FUNCTION_BLOCK EC_SENSORS_ACTUATORS (* Composite Function Block Type *)
  (* Standard: 61499-2 *)
  (* Version 1.0, 2019-03-30, adeel *)
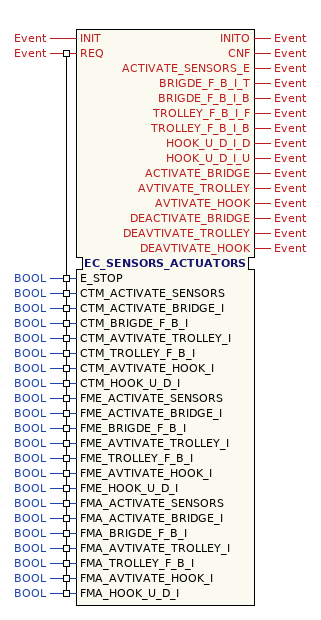
  EVENT_INPUT
    INIT; (* Initialization Request *)
    REQ WITH CTM_ACTIVATE_SENSORS, CTM_ACTIVATE_BRIDGE_I, CTM_BRIGDE_F_B_I, CTM_AVTIVATE_TROLLEY_I, CTM_TROLLEY_F_B_I, CTM_AVTIVATE_HOOK_I, CTM_HOOK_U_D_I, FME_ACTIVATE_SENSORS, FME_ACTIVATE_BRIDGE_I, FME_BRIGDE_F_B_I, FME_AVTIVATE_TROLLEY_I, FME_TROLLEY_F_B_I, FME_AVTIVATE_HOOK_I, FME_HOOK_U_D_I, FMA_ACTIVATE_SENSORS, FMA_ACTIVATE_BRIDGE_I, FMA_BRIGDE_F_B_I, FMA_AVTIVATE_TROLLEY_I, FMA_TROLLEY_F_B_I, FMA_AVTIVATE_HOOK_I, FMA_HOOK_U_D_I, E_STOP; (* Normal Execution Request *)
  END_EVENT
  EVENT_OUTPUT
    INITO; (* Initialization Confirm *)
    CNF;
    ACTIVATE_SENSORS_E;
    BRIGDE_F_B_I_T;
    BRIGDE_F_B_I_B;
    TROLLEY_F_B_I_F;
    TROLLEY_F_B_I_B;
    HOOK_U_D_I_D;
    HOOK_U_D_I_U;
    ACTIVATE_BRIDGE;
    AVTIVATE_TROLLEY;
    AVTIVATE_HOOK;
    DEACTIVATE_BRIDGE;
    DEAVTIVATE_TROLLEY;
    DEAVTIVATE_HOOK;
  END_EVENT
  VAR_INPUT
    E_STOP : BOOL;
    CTM_ACTIVATE_SENSORS : BOOL;
    CTM_ACTIVATE_BRIDGE_I : BOOL;
    CTM_BRIGDE_F_B_I : BOOL;
    CTM_AVTIVATE_TROLLEY_I : BOOL;
    CTM_TROLLEY_F_B_I : BOOL;
    CTM_AVTIVATE_HOOK_I : BOOL;
    CTM_HOOK_U_D_I : BOOL;
    FME_ACTIVATE_SENSORS : BOOL;
    FME_ACTIVATE_BRIDGE_I : BOOL;
    FME_BRIGDE_F_B_I : BOOL;
    FME_AVTIVATE_TROLLEY_I : BOOL;
    FME_TROLLEY_F_B_I : BOOL;
    FME_AVTIVATE_HOOK_I : BOOL;
    FME_HOOK_U_D_I : BOOL;
    FMA_ACTIVATE_SENSORS : BOOL;
    FMA_ACTIVATE_BRIDGE_I : BOOL;
    FMA_BRIGDE_F_B_I : BOOL;
    FMA_AVTIVATE_TROLLEY_I : BOOL;
    FMA_TROLLEY_F_B_I : BOOL;
    FMA_AVTIVATE_HOOK_I : BOOL;
    FMA_HOOK_U_D_I : BOOL;
  END_VAR
  FBS
    CTM_11 : E_R_TRIG;
    CTM_12 : E_F_TRIG;
    CTM_21 : E_R_TRIG;
    CTM_22 : E_F_TRIG;
    CTM_31 : E_R_TRIG;
    CTM_32 : E_F_TRIG;
    CTM_41 : E_R_TRIG;
    CTM_42 : E_F_TRIG;
    FME41 : E_R_TRIG;
    FME_11 : E_R_TRIG;
    FME_32 : E_F_TRIG;
    FME_42 : E_F_TRIG;
    FME_31 : E_R_TRIG;
    FME_12 : E_F_TRIG;
    FME_21 : E_R_TRIG;
    FME_22 : E_F_TRIG;
    FMA_41 : E_R_TRIG;
    FMA_11 : E_R_TRIG;
    FMA_32 : E_F_TRIG;
    FMA_42 : E_F_TRIG;
    FMA_31 : E_R_TRIG;
    FMA_12 : E_F_TRIG;
    FMA_21 : E_R_TRIG;
    FMA_22 : E_F_TRIG;
    E_CYCLE : E_CYCLE(DT := T#100ms);
    E_CYCLE_1 : E_CYCLE(DT := T#100ms);
    E_CYCLE_2 : E_CYCLE(DT := T#100ms);
    HA_CTM : E_R_TRIG;
    BA_CTM : E_R_TRIG;
    TA_FME : E_R_TRIG;
    BA_FMA : E_R_TRIG;
    TA_CTM : E_R_TRIG;
    BA_FME : E_R_TRIG;
    HA_FME : E_R_TRIG;
    TA_FMA : E_R_TRIG;
    HA_FMA : E_R_TRIG;
    BD_CTM : E_F_TRIG;
    TD_CTM : E_F_TRIG;
    HD_CTM : E_F_TRIG;
    BD_FME : E_F_TRIG;
    TD_FME : E_F_TRIG;
    HD_FME : E_F_TRIG;
    BD_FMA : E_F_TRIG;
    TD_FMA : E_F_TRIG;
    HD_FMA : E_F_TRIG;
    E_STOP : E_F_TRIG;
    E_F_TRIG : E_F_TRIG;
  END_FBS
  EVENT_CONNECTIONS
    E_CYCLE.EO TO ACTIVATE_SENSORS_E;
    E_CYCLE_1.EO TO ACTIVATE_SENSORS_E;
    E_CYCLE_2.EO TO ACTIVATE_SENSORS_E;
    CTM_11.EO TO E_CYCLE.START;
    CTM_12.EO TO E_CYCLE.STOP;
    INIT TO INITO;
    FME_11.EO TO E_CYCLE_1.START;
    FME_12.EO TO E_CYCLE_1.STOP;
    FMA_11.EO TO E_CYCLE_2.START;
    FMA_12.EO TO E_CYCLE_2.STOP;
    REQ TO CTM_11.EI;
    REQ TO CTM_12.EI;
    REQ TO FME_11.EI;
    REQ TO FME_12.EI;
    REQ TO FMA_11.EI;
    REQ TO FMA_12.EI;
    REQ TO CNF;
    REQ TO CTM_21.EI;
    REQ TO CTM_22.EI;
    CTM_21.EO TO BRIGDE_F_B_I_T;
    CTM_22.EO TO BRIGDE_F_B_I_B;
    REQ TO CTM_31.EI;
    REQ TO CTM_32.EI;
    CTM_31.EO TO TROLLEY_F_B_I_F;
    CTM_32.EO TO TROLLEY_F_B_I_B;
    REQ TO CTM_41.EI;
    REQ TO CTM_42.EI;
    CTM_41.EO TO HOOK_U_D_I_D;
    CTM_42.EO TO HOOK_U_D_I_U;
    REQ TO FME_21.EI;
    REQ TO FME_22.EI;
    REQ TO FME_31.EI;
    REQ TO FME_32.EI;
    REQ TO FME41.EI;
    REQ TO FME_42.EI;
    FME_21.EO TO BRIGDE_F_B_I_T;
    FME_22.EO TO BRIGDE_F_B_I_B;
    FME_31.EO TO TROLLEY_F_B_I_F;
    FME_32.EO TO TROLLEY_F_B_I_B;
    FME41.EO TO HOOK_U_D_I_D;
    FME_42.EO TO HOOK_U_D_I_U;
    FMA_21.EO TO BRIGDE_F_B_I_T;
    FMA_22.EO TO BRIGDE_F_B_I_B;
    FMA_31.EO TO TROLLEY_F_B_I_F;
    FMA_32.EO TO TROLLEY_F_B_I_B;
    FMA_41.EO TO HOOK_U_D_I_D;
    FMA_42.EO TO HOOK_U_D_I_U;
    REQ TO FMA_21.EI;
    REQ TO FMA_22.EI;
    REQ TO FMA_31.EI;
    REQ TO FMA_32.EI;
    REQ TO FMA_41.EI;
    REQ TO FMA_42.EI;
    BA_CTM.EO TO ACTIVATE_BRIDGE;
    BA_FME.EO TO ACTIVATE_BRIDGE;
    BA_FMA.EO TO ACTIVATE_BRIDGE;
    TA_CTM.EO TO AVTIVATE_TROLLEY;
    TA_FME.EO TO AVTIVATE_TROLLEY;
    TA_FMA.EO TO AVTIVATE_TROLLEY;
    HA_CTM.EO TO AVTIVATE_HOOK;
    HA_FME.EO TO AVTIVATE_HOOK;
    HA_FMA.EO TO AVTIVATE_HOOK;
    REQ TO BA_CTM.EI;
    REQ TO TA_CTM.EI;
    REQ TO HA_CTM.EI;
    REQ TO BA_FME.EI;
    REQ TO TA_FME.EI;
    REQ TO HA_FME.EI;
    REQ TO BA_FMA.EI;
    REQ TO TA_FMA.EI;
    REQ TO HA_FMA.EI;
    BD_CTM.EO TO DEACTIVATE_BRIDGE;
    BD_FME.EO TO DEACTIVATE_BRIDGE;
    BD_FMA.EO TO DEACTIVATE_BRIDGE;
    TD_CTM.EO TO DEAVTIVATE_TROLLEY;
    TD_FME.EO TO DEAVTIVATE_TROLLEY;
    TD_FMA.EO TO DEAVTIVATE_TROLLEY;
    HD_CTM.EO TO DEAVTIVATE_HOOK;
    REQ TO BD_CTM.EI;
    REQ TO TD_CTM.EI;
    REQ TO HD_CTM.EI;
    REQ TO BD_FME.EI;
    REQ TO TD_FME.EI;
    REQ TO HD_FME.EI;
    REQ TO BD_FMA.EI;
    REQ TO TD_FMA.EI;
    REQ TO HD_FMA.EI;
    REQ TO E_STOP.EI;
    E_STOP.EO TO DEACTIVATE_BRIDGE;
    E_STOP.EO TO DEAVTIVATE_TROLLEY;
    E_F_TRIG.EO TO E_CYCLE.STOP;
    E_F_TRIG.EO TO E_CYCLE_1.STOP;
    E_F_TRIG.EO TO E_CYCLE_2.STOP;
    REQ TO E_F_TRIG.EI;
  END_CONNECTIONS
  DATA_CONNECTIONS
    CTM_ACTIVATE_SENSORS TO CTM_11.QI;
    CTM_ACTIVATE_SENSORS TO CTM_12.QI;
    FME_ACTIVATE_SENSORS TO FME_11.QI;
    FME_ACTIVATE_SENSORS TO FME_12.QI;
    FMA_ACTIVATE_SENSORS TO FMA_11.QI;
    FMA_ACTIVATE_SENSORS TO FMA_12.QI;
    CTM_BRIGDE_F_B_I TO CTM_21.QI;
    CTM_BRIGDE_F_B_I TO CTM_22.QI;
    CTM_TROLLEY_F_B_I TO CTM_31.QI;
    CTM_TROLLEY_F_B_I TO CTM_32.QI;
    CTM_HOOK_U_D_I TO CTM_41.QI;
    CTM_HOOK_U_D_I TO CTM_42.QI;
    FME_BRIGDE_F_B_I TO FME_21.QI;
    FME_BRIGDE_F_B_I TO FME_22.QI;
    FME_TROLLEY_F_B_I TO FME_31.QI;
    FME_TROLLEY_F_B_I TO FME_32.QI;
    FME_HOOK_U_D_I TO FME41.QI;
    FME_HOOK_U_D_I TO FME_42.QI;
    FMA_BRIGDE_F_B_I TO FMA_21.QI;
    FMA_BRIGDE_F_B_I TO FMA_22.QI;
    FMA_TROLLEY_F_B_I TO FMA_31.QI;
    FMA_TROLLEY_F_B_I TO FMA_32.QI;
    FMA_HOOK_U_D_I TO FMA_41.QI;
    FMA_HOOK_U_D_I TO FMA_42.QI;
    CTM_ACTIVATE_BRIDGE_I TO BA_CTM.QI;
    CTM_AVTIVATE_TROLLEY_I TO TA_CTM.QI;
    CTM_AVTIVATE_HOOK_I TO HA_CTM.QI;
    FME_ACTIVATE_BRIDGE_I TO BA_FME.QI;
    FME_AVTIVATE_TROLLEY_I TO TA_FME.QI;
    FME_AVTIVATE_HOOK_I TO HA_FME.QI;
    FMA_ACTIVATE_BRIDGE_I TO BA_FMA.QI;
    FMA_AVTIVATE_TROLLEY_I TO TA_FMA.QI;
    FMA_AVTIVATE_HOOK_I TO HA_FMA.QI;
    CTM_AVTIVATE_TROLLEY_I TO TD_CTM.QI;
    CTM_AVTIVATE_HOOK_I TO HD_CTM.QI;
    FME_ACTIVATE_BRIDGE_I TO BD_FME.QI;
    FME_AVTIVATE_TROLLEY_I TO TD_FME.QI;
    FME_AVTIVATE_HOOK_I TO HD_FME.QI;
    FMA_ACTIVATE_BRIDGE_I TO BD_FMA.QI;
    FMA_AVTIVATE_TROLLEY_I TO TD_FMA.QI;
    FMA_AVTIVATE_HOOK_I TO HD_FMA.QI;
    E_STOP TO E_STOP.QI;
    CTM_ACTIVATE_BRIDGE_I TO BD_CTM.QI;
    E_STOP TO E_F_TRIG.QI;
  END_CONNECTIONS
END_FUNCTION_BLOCK
